FUNCTION_BLOCK ABSTRACT FB_Conveyor
VAR_INPUT
    // Machine control
    stMachineControl: ST_MachineControl;
END_VAR
VAR_OUTPUT
    // Output to conveyor motor
    bConveyorOn: BOOL;
END_VAR
VAR
    // Part moving timeout
    fbMovingTimeout: TON;
    // Run-down-timeout after normal stop
    fbRunDownTimeout: TOF;
    // Current state of conveyor
    eStateConveyor: (C_IDLE, C_RUNNING, C_RUNNING_OUT, C_LOCKOUT);
END_VAR

// Cyclic call of timer for moving timeout in derived function block
IF fbMovingTimeout.PT > T#0S THEN
    fbMovingTimeout();
END_IF

// Cyclic call of timer for run-down-timeout after normal stop
IF fbRunDownTimeout.PT > T#0S THEN
    fbRunDownTimeout();
END_IF

// Emergency stop is active
IF NOT stMachineControl.bEmergStopNC THEN
    eStateConveyor := C_LOCKOUT;
END_IF


CASE eStateConveyor OF
    C_IDLE:
        bConveyorOn := FALSE;
        fbRunDownTimeout.IN := FALSE;

    C_RUNNING:
        bConveyorOn := TRUE;
        fbRunDownTimeout.IN := TRUE;

    C_RUNNING_OUT:
        fbRunDownTimeout.IN := FALSE;
        IF NOT fbRunDownTimeout.Q OR fbRunDownTimeout.PT = T#0S THEN
            eStateConveyor := C_IDLE;
        END_IF

    C_LOCKOUT:
        bConveyorOn := FALSE;
        fbRunDownTimeout.IN := FALSE;
END_CASE

METHOD PUBLIC Reset
VAR_INPUT
END_VAR
IF stMachineControl.bEmergStopNC AND eStateConveyor = C_LOCKOUT THEN
    eStateConveyor := C_IDLE;
END_IF
END_METHOD

METHOD PROTECTED Start
VAR_INPUT
END_VAR
IF eStateConveyor = C_IDLE OR eStateConveyor = C_RUNNING_OUT THEN
    eStateConveyor := C_RUNNING;
END_IF
END_METHOD

METHOD PROTECTED Stop
VAR_INPUT
    // Enable timeout before conveyor halt
    bRunOut: BOOL := FALSE;
END_VAR
IF eStateConveyor = C_RUNNING THEN
    // Stop converyor with timeout before halt
    IF fbRunDownTimeout.PT > T#0S AND bRunOut THEN
        eStateConveyor := C_RUNNING_OUT;

    // Stop conveyor immediately
    ELSE
        eStateConveyor := C_IDLE;
    END_IF
END_IF
END_METHOD

// Part moving timeout
{attribute 'monitoring' := 'call'}
PROPERTY PUBLIC tMovingTimeout: TIME
GET
tMovingTimeout := fbMovingTimeout.PT;
END_GET
SET
fbMovingTimeout.PT := tMovingTimeout;
END_SET
END_PROPERTY

// Run-down-timeout after normal stop
{attribute 'monitoring' := 'call'}
PROPERTY PUBLIC tRunDownTimeout: TIME
GET
tRunDownTimeout := fbRunDownTimeout.PT;
END_GET
SET
fbRunDownTimeout.PT := tRunDownTimeout;
END_SET
END_PROPERTY

END_FUNCTION_BLOCK

(* stored: Version 1.1.0.1
   POU FB_Conveyor: Id {245a5808-fce9-4686-b31f-3aa50bc94906}, SpecialFunc None
   Method Reset: Id {c6f9219d-30dc-4aaa-a52b-80bf5ad63bc8}
   Method Start: Id {e5324438-ffcb-4c49-a5d6-8babf4557efa}
   Method Stop: Id {497f56fe-7509-4e86-b27b-bdcc17baac39}
   Property tMovingTimeout: Id {d6846ea9-b660-4c68-926b-4c307d706c12}
   Get Get: Id {ef2e8eb8-38a9-4c47-a0e6-f0b2558ec260}
   Set Set: Id {37f62f04-9445-4ecc-aab4-6c0bc2cfc248}
   Property tRunDownTimeout: Id {4b764709-8d3d-4944-95b7-04a2d130102e}
   Get Get: Id {245e477e-a008-409d-aec7-abdc2592ce40}
   Set Set: Id {5476210a-bee1-4eef-b655-9d8c659c6410} *)
